Fanuc KAREL source: KA00014.KL

PROGRAM KA00014
%NOLOCKGROUP
VAR
  SRC: REAL
  DST: REAL
BEGIN
  SRC = 2.0
  DST = SRC
END KA00014
